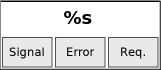
VISUALIZATION vSensorFrame  // 161x70
VAR_INPUT
		iNameIndex :INT;
END_VAR
VAR_IN_OUT
	fbSensor :FB_Sensor;

END_VAR
    Rectangle (0,1 161x69)
    Rectangle (2,37 50x30), "Signal", colour toggle: fbSensor.bSensorSignal
    Rectangle (108,37 50x30), "Req.", colour toggle: fbSensor.bRequestedState
    Rectangle (55,37 50x30), "Error", colour toggle: fbSensor.prSensorOnError OR fbSensor.prSensorOffError
    Rectangle (3,3 150x30), "%s", text list: 'tlSensorNames', text index: iNameIndex
END_VISUALIZATION

(* stored: Version 1.1.0.1, ProductVersion 3.1.4024.15
   Visu vSensorFrame: Id {cbf39ea4-9e6c-4591-ada2-89e11b647e28} *)
